PROGRAM F15_AS3_MQ41
VAR
	Energimatare: FB_SCHNEIDER_iEM3150;
	tof_0: TOF;

	FB_FL0: FB_FL;
END_VAR


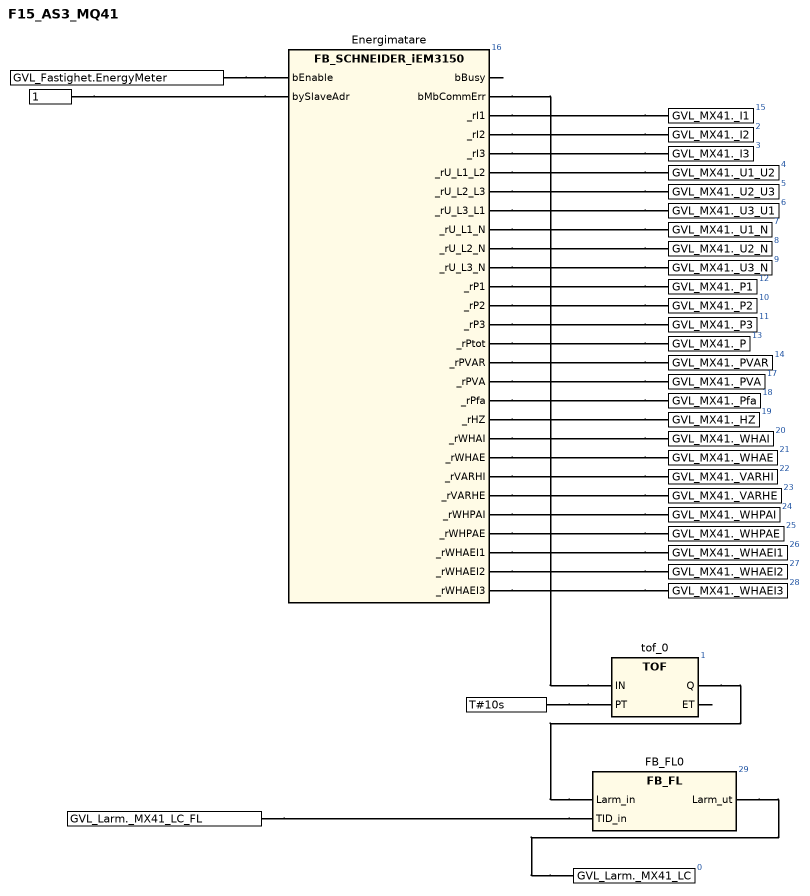
// PAGE
GVL_Larm._MX41_LC := FB_FL0.Larm_ut;
tof_0(IN := Energimatare.bMbCommErr, PT := T#10s); // TOF
GVL_MX41._I2 := Energimatare._rI2;
GVL_MX41._I3 := Energimatare._rI3;
GVL_MX41._U1_U2 := Energimatare._rU_L1_L2;
GVL_MX41._U2_U3 := Energimatare._rU_L2_L3;
GVL_MX41._U3_U1 := Energimatare._rU_L3_L1;
GVL_MX41._U1_N := Energimatare._rU_L1_N;
GVL_MX41._U2_N := Energimatare._rU_L2_N;
GVL_MX41._U3_N := Energimatare._rU_L3_N;
GVL_MX41._P2 := Energimatare._rP2;
GVL_MX41._P3 := Energimatare._rP3;
GVL_MX41._P1 := Energimatare._rP1;
GVL_MX41._P := Energimatare._rPtot;
GVL_MX41._PVAR := Energimatare._rPVAR;
GVL_MX41._I1 := Energimatare._rI1;
Energimatare(bEnable := GVL_Fastighet.EnergyMeter, bySlaveAdr := 1); // FB_SCHNEIDER_iEM3150
GVL_MX41._PVA := Energimatare._rPVA;
GVL_MX41._Pfa := Energimatare._rPfa;
GVL_MX41._HZ := Energimatare._rHZ;
GVL_MX41._WHAI := Energimatare._rWHAI;
GVL_MX41._WHAE := Energimatare._rWHAE;
GVL_MX41._VARHI := Energimatare._rVARHI;
GVL_MX41._VARHE := Energimatare._rVARHE;
GVL_MX41._WHPAI := Energimatare._rWHPAI;
GVL_MX41._WHPAE := Energimatare._rWHPAE;
GVL_MX41._WHAEI1 := Energimatare._rWHAEI1;
GVL_MX41._WHAEI2 := Energimatare._rWHAEI2;
GVL_MX41._WHAEI3 := Energimatare._rWHAEI3;
FB_FL0(Larm_in := tof_0.Q, TID_in := GVL_Larm._MX41_LC_FL); // FB_FL

END_PROGRAM

(* stored: Version 1.1.0.1, ProductVersion 3.1.4022.3
   POU F15_AS3_MQ41: Id {8ab68090-1f8b-4507-a6ea-15cfb72f29cb}, SpecialFunc None *)
